TYPE ST_HMI_HoneywellStatus :
STRUCT

(* read only *)
	bHandScanerPortOK			: BOOL;
	bHandScannerBaudrateOK	: BOOL;
	sLastScannerBarcode		: T_MaxString;

END_STRUCT
END_TYPE

(* stored: Version 1.1.0.1, ProductVersion 3.1.4024.15
   DUT ST_HMI_HoneywellStatus: Id {b26faea6-bcc1-43a7-8192-fa45b78bdd68} *)
